% RSLogix 500 project THREE-PHASE MOTOR CONTROL F-R 3PB DIR CHNG.RSS, saved by version 10.00.00.00 %
PROJECT "MRLEIGH"    % processor: Bul.1763 MicroLogix 1100 Series B %

PROGRAM FILES
  LAD 2 "MAIN"  15 rungs  % Invert Signals Wired Failsafe %

DATA FILES
  O0 OUTPUT  4 elements
  I1 INPUT  6 elements
  S2 STATUS  66 elements
  B3 BINARY  1 elements
  T4 TIMER  1 elements
  C5 COUNTER  1 elements
  R6 CONTROL  1 elements
  N7 INTEGER  1 elements
  F8 FLOAT  1 elements

LADDER 2 "MAIN"    % Invert Signals Wired Failsafe %
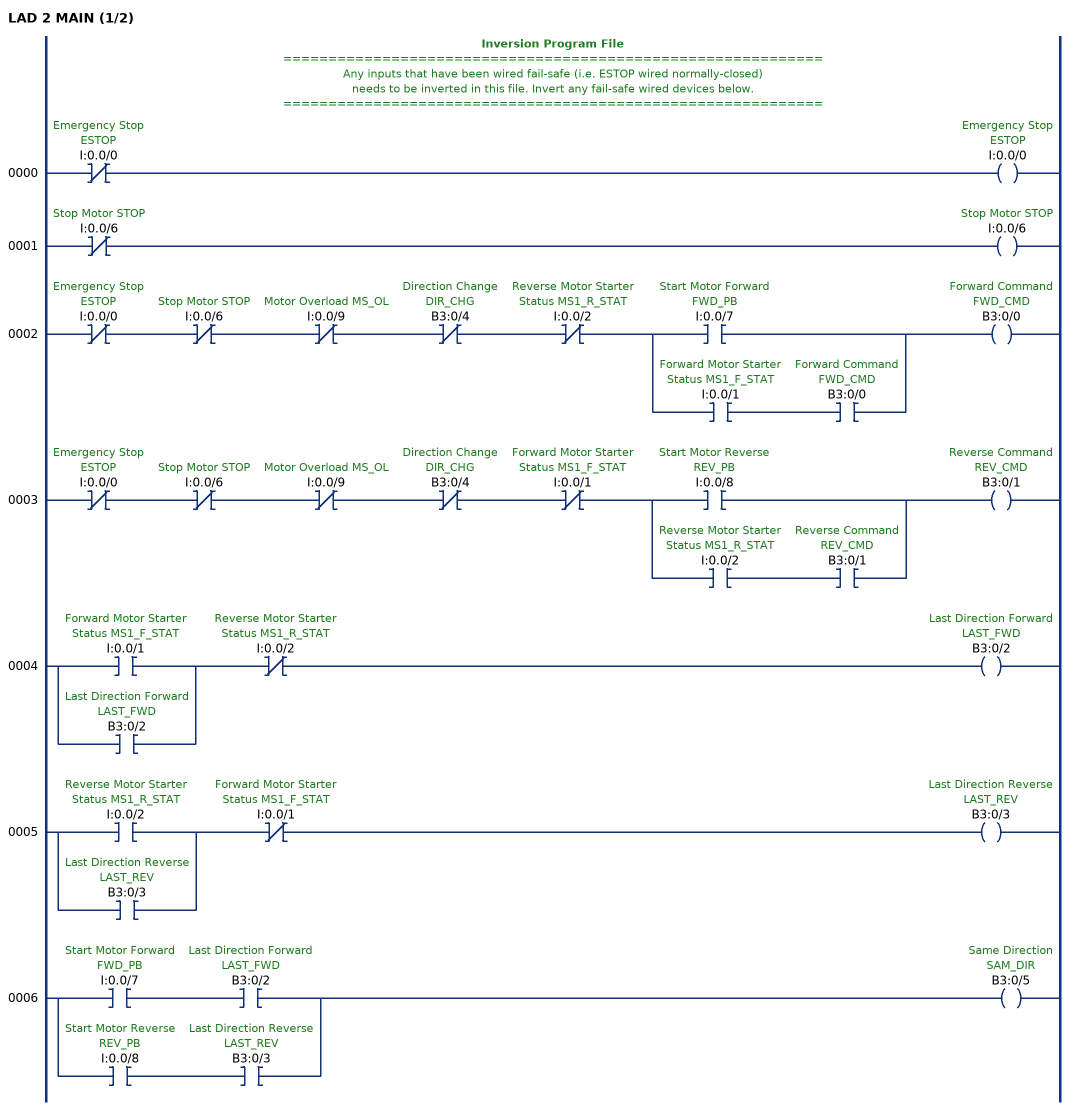
% Rung: 0 %
% TITLE: Inversion Program File %
% ============================================================
% 
%   Any inputs that have been wired fail-safe (i.e. ESTOP wired normally-closed)
%   needs to be inverted in this file. Invert any fail-safe wired devices below.
% 
% ============================================================ %
SOR XIO I:0.0/0 OTE I:0.0/0 EOR
%   I:0.0/0  ESTOP  "Emergency Stop" %
% Rung: 1 %
SOR XIO I:0.0/6 OTE I:0.0/6 EOR
%   I:0.0/6  STOP  "Stop Motor" %
% Rung: 2 %
SOR XIO I:0.0/0 XIO I:0.0/6 XIO I:0.0/9 XIO B3:0/4 XIO I:0.0/2 BST XIC I:0.0/7 NXB XIC I:0.0/1 XIC B3:0/0 BND OTE B3:0/0 EOR
%   I:0.0/0  ESTOP  "Emergency Stop" %
%   I:0.0/6  STOP  "Stop Motor" %
%   I:0.0/9  MS_OL  "Motor Overload" %
%   B3:0/4  DIR_CHG  "Direction Change" %
%   I:0.0/2  MS1_R_STAT  "Reverse Motor Starter Status" %
%   I:0.0/7  FWD_PB  "Start Motor Forward" %
%   I:0.0/1  MS1_F_STAT  "Forward Motor Starter Status" %
%   B3:0/0  FWD_CMD  "Forward Command" %
% Rung: 3 %
SOR XIO I:0.0/0 XIO I:0.0/6 XIO I:0.0/9 XIO B3:0/4 XIO I:0.0/1 BST XIC I:0.0/8 NXB XIC I:0.0/2 XIC B3:0/1 BND OTE B3:0/1 EOR
%   I:0.0/0  ESTOP  "Emergency Stop" %
%   I:0.0/6  STOP  "Stop Motor" %
%   I:0.0/9  MS_OL  "Motor Overload" %
%   B3:0/4  DIR_CHG  "Direction Change" %
%   I:0.0/1  MS1_F_STAT  "Forward Motor Starter Status" %
%   I:0.0/8  REV_PB  "Start Motor Reverse" %
%   I:0.0/2  MS1_R_STAT  "Reverse Motor Starter Status" %
%   B3:0/1  REV_CMD  "Reverse Command" %
% Rung: 4 %
SOR BST XIC I:0.0/1 NXB XIC B3:0/2 BND XIO I:0.0/2 OTE B3:0/2 EOR
%   I:0.0/1  MS1_F_STAT  "Forward Motor Starter Status" %
%   B3:0/2  LAST_FWD  "Last Direction Forward" %
%   I:0.0/2  MS1_R_STAT  "Reverse Motor Starter Status" %
% Rung: 5 %
SOR BST XIC I:0.0/2 NXB XIC B3:0/3 BND XIO I:0.0/1 OTE B3:0/3 EOR
%   I:0.0/2  MS1_R_STAT  "Reverse Motor Starter Status" %
%   B3:0/3  LAST_REV  "Last Direction Reverse" %
%   I:0.0/1  MS1_F_STAT  "Forward Motor Starter Status" %
% Rung: 6 %
SOR BST XIC I:0.0/7 XIC B3:0/2 NXB XIC I:0.0/8 XIC B3:0/3 BND OTE B3:0/5 EOR
%   I:0.0/7  FWD_PB  "Start Motor Forward" %
%   B3:0/2  LAST_FWD  "Last Direction Forward" %
%   I:0.0/8  REV_PB  "Start Motor Reverse" %
%   B3:0/3  LAST_REV  "Last Direction Reverse" %
%   B3:0/5  SAM_DIR  "Same Direction" %

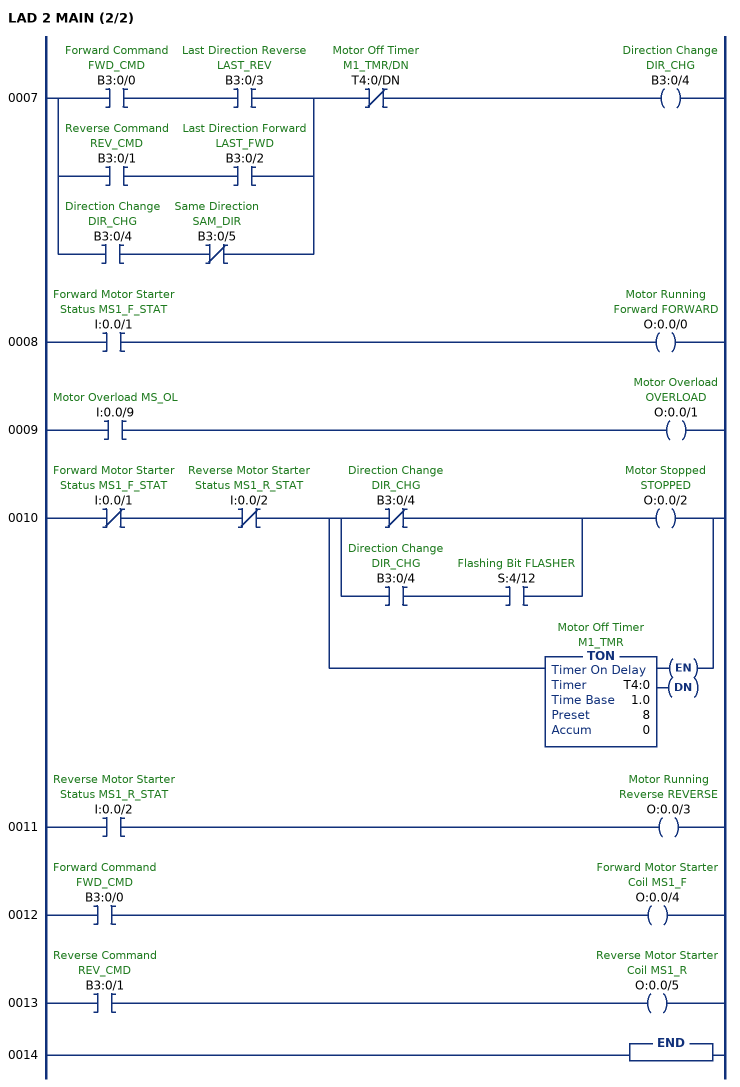
% Rung: 7 %
SOR BST XIC B3:0/0 XIC B3:0/3 NXB XIC B3:0/1 XIC B3:0/2 NXB XIC B3:0/4 XIO B3:0/5 BND XIO T4:0/DN OTE B3:0/4 EOR
%   B3:0/0  FWD_CMD  "Forward Command" %
%   B3:0/3  LAST_REV  "Last Direction Reverse" %
%   B3:0/1  REV_CMD  "Reverse Command" %
%   B3:0/2  LAST_FWD  "Last Direction Forward" %
%   B3:0/4  DIR_CHG  "Direction Change" %
%   B3:0/5  SAM_DIR  "Same Direction" %
%   T4:0  M1_TMR  "Motor Off Timer" %
% Rung: 8 %
SOR XIC I:0.0/1 OTE O:0.0/0 EOR
%   I:0.0/1  MS1_F_STAT  "Forward Motor Starter Status" %
%   O:0.0/0  FORWARD  "Motor Running Forward" %
% Rung: 9 %
SOR XIC I:0.0/9 OTE O:0.0/1 EOR
%   I:0.0/9  MS_OL  "Motor Overload" %
%   O:0.0/1  OVERLOAD  "Motor Overload" %
% Rung: 10 %
SOR XIO I:0.0/1 XIO I:0.0/2 BST BST XIO B3:0/4 NXB XIC B3:0/4 XIC S:4/12 BND OTE O:0.0/2 NXB TON T4:0 1.0 8 0 BND EOR
%   I:0.0/1  MS1_F_STAT  "Forward Motor Starter Status" %
%   I:0.0/2  MS1_R_STAT  "Reverse Motor Starter Status" %
%   B3:0/4  DIR_CHG  "Direction Change" %
%   S:4/12  FLASHER  "Flashing Bit" %
%   O:0.0/2  STOPPED  "Motor Stopped" %
%   T4:0  M1_TMR  "Motor Off Timer" %
% Rung: 11 %
SOR XIC I:0.0/2 OTE O:0.0/3 EOR
%   I:0.0/2  MS1_R_STAT  "Reverse Motor Starter Status" %
%   O:0.0/3  REVERSE  "Motor Running Reverse" %
% Rung: 12 %
SOR XIC B3:0/0 OTE O:0.0/4 EOR
%   B3:0/0  FWD_CMD  "Forward Command" %
%   O:0.0/4  MS1_F  "Forward Motor Starter Coil" %
% Rung: 13 %
SOR XIC B3:0/1 OTE O:0.0/5 EOR
%   B3:0/1  REV_CMD  "Reverse Command" %
%   O:0.0/5  MS1_R  "Reverse Motor Starter Coil" %
% Rung: 14 %
SOR END EOR

OTHER DOCUMENTED ADDRESSES
  B3:0/15  GOOD  "All Disablers Good"
  I:0.0/3  FWD_SS  "Forward Selection"
  I:0.0/4  REV_SS  "Reverse Selection"
  PFILE:3  "Simulation"
  PFILE:4  "Main Program"
  U:3  SIM  "Simulation Program File"
  U:4  MAIN  "Main Program File"

DATA TABLE (non-zero values as saved)
DATA T4
% .PRE .ACC %
% T4:0 % 8 0
